ABB RobotStudio station: JogRobot_20211110-171003.rsstn

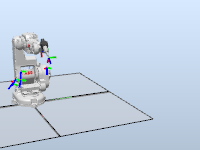
Station JogRobot (saved by RobotStudio 21.2.9526.0)
Controller CRB1100_4_47_Controller
  mechanical unit ROB_1: IRB140_6_81_C_03, 6 joints, base frame (0, 0, 0) mm
Layout (positions relative to the parent item):
  - IRB140_6_81_C_03 [mechanism, from Robots\IRB140_6_81_C_G_03.rslib] at (0, 0, 0) mm; joint values [0, 0, 0, 0, 0, 0] (rad or m)
  - MyTool [mechanism, from Training Objects\myTool.rslib] at (515, 0, 712) mm, rotated rx 0 ry 90 rz 0 deg
Attachment: MyTool is attached to IRB140_6_81_C_03 / Link6
Targets, tools, work objects and paths stored in the station, written as RAPID:
! task T_ROB1
MODULE CalibData
  PERS tooldata MyTool:=[TRUE,[[31.792631019,0,229.638935148],[0.945518576,0,0.325568154,0]],[1,[0,0,1],[1,0,0,0],0,0,0]];
ENDMODULE

! task T_ROB1
MODULE Module1
  CONST robtarget Target_10:=[[744.638935148,0,680.207368981],[0.438371147,0,0.898794046,0],[0,0,0,0],[9E+09,9E+09,9E+09,9E+09,9E+09,9E+09]];
  CONST robtarget Target_20:=[[684.912746939,-249.287852955,563.540548812],[0.352923536,0.16211454,0.919397242,-0.062229941],[-1,0,-1,0],[9E+09,9E+09,9E+09,9E+09,9E+09,9E+09]];
  CONST robtarget Target_30:=[[626.484387754,-285.791516778,484.136304693],[0.116814872,-0.010012123,0.942233983,-0.313766097],[-1,-1,-1,0],[9E+09,9E+09,9E+09,9E+09,9E+09,9E+09]];
  CONST robtarget Target_40:=[[550.156869486,-296.399513088,423.891813595],[0.08708963,0.135558162,-0.917937518,0.362532887],[-1,-1,-1,0],[9E+09,9E+09,9E+09,9E+09,9E+09,9E+09]];
  CONST robtarget Target_50:=[[639.457437944,-244.315037455,472.821458625],[0.162298125,0.055675429,0.971810102,-0.161693199],[-1,-1,-1,0],[9E+09,9E+09,9E+09,9E+09,9E+09,9E+09]];
  CONST robtarget Target_60:=[[716.652078506,-10.873720218,583.1539495],[0.271449806,-0.102067838,0.946657971,-0.140484327],[0,-1,-1,0],[9E+09,9E+09,9E+09,9E+09,9E+09,9E+09]];
  CONST robtarget Target_70:=[[744.638935148,0,680.207368981],[0.438371147,0,0.898794046,0],[0,0,0,0],[9E+09,9E+09,9E+09,9E+09,9E+09,9E+09]];
ENDMODULE

